# EPICS autosave request: ipApp/Db/HG-100_settings.req
$(P)$(R)Temperature
$(P)$(R)Slope
$(P)$(R)Offset
